// TIA Portal V17 export
// export: Created 2025-01-16T19:22:27.1780597Z, ExportSetting WithDefaults, DisplayName Totally Integrated Automation Portal, DisplayVersion V17 Update 6, DisplayName TIA Portal Openness, DisplayVersion V17 Update 6, DisplayName TIA Portal Version Control Interface, DisplayVersion V17, DisplayName STEP 7 Professional, DisplayVersion V17 Update 6, DisplayName STEP 7 Safety, DisplayVersion V17 Update 6, DisplayName WinCC Advanced, DisplayVersion V17 Update 6
ORGANIZATION_BLOCK "Main"   // OB1, LAD, ProgramCycle
TITLE = "Main Program Sweep (Cycle)"
{ S7_Optimized_Access := 'TRUE' }
VERSION : 0.1
// stored: AutoNumber true, IsIECCheckEnabled false, SetENOAutomatically false
   VAR_INPUT
      Initial_Call : Bool;   // Initial call of this OB
      Remanence : Bool;   // =True, if remanent data are available
   END_VAR
BEGIN

REGION Network 1
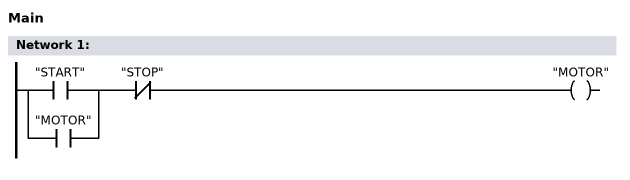
   RUNG wire#powerrail
      Contact( "START" )
      wire#w1
      I_Contact( "STOP" )
      Coil( "MOTOR" )
   END_RUNG
   RUNG wire#powerrail
      Contact( "MOTOR" )
   END_RUNG wire#w1
   // the same network as SCL:
   "MOTOR" := ("START" OR "MOTOR") AND NOT "STOP";
END_REGION
END_ORGANIZATION_BLOCK
